KUKA KRL program: RobotSps.src, robotsps.dat

--- RobotSps.src ---
&ACCESS RVE
&REL 156
&COMMENT Ansteuerung Micromaster Frequenzumrichter
&PARAM EDITMASK = *
&PARAM TEMPLATE = C:\KRC\Roboter\Template\ExpertSubmit
DEF RobotSps( )

;************************************************
;              CNC Robotics Ltd
;              www.cncrobotics.co.uk
;************************************************
;     Contact: helpdesk@cncrobotics.co.uk
;     Date: 12/09/23
;     Version: 0.23.48
;************************************************
; Description: sps control specific for the spindle.
;************************************************




IF $T1 THEN
   oMode = 0;
ENDIF
IF $T2 THEN
   oMode = 1;
ENDIF
IF $AUT THEN
   oMode = 2;
ENDIF
IF $EXT THEN
   oMode = 3;
ENDIF

bDoorFault = ($AUT OR $EXT) AND (NOT iDoorSignal)

END

--- robotsps.dat ---
&ACCESS  RV
&COMMENT Ansteuerung Micromaster Frequenzumrichter
&PARAM EDITMASK = *
&PARAM TEMPLATE = C:\KRC\Roboter\Template\ExpertSubmit
&PARAM TEMPLATE = C:\KRC\Roboter\Template\ExpertSubmit
&REL 156
DEFDAT  ROBOTSPS PUBLIC
GLOBAL INT nHeartbeatTime=-1000

;digital inputs

;GLOBAL SIGNAL iDrivesEnabled $IN[] ;drive engage from Pilz mapped directly by Auto External;
;GLOBAL SIGNAL iAcknowledgeMessages $IN[] ;Acknowledge messages from Pilz mapped directly by Auto External
;GLOBAL SIGNAL iStart $IN[] ;operator start button
;GLOBAL SIGNAL iStop $IN[] ;operator stop button
;
;GLOBAL SIGNAL oTeach $OUT[] ;T1 active to Pilz


GLOBAL ENUM SYSTEM_STATE EMERGENCY_STOP,DOOR_OPEN,FAULT,SYSTEM_OK,DRIVES_ON
DECL GLOBAL SYSTEM_STATE systemState=#SYSTEM_OK
DECL GLOBAL STATE_T E_stat
DECL GLOBAL MODUS_T E_mode
GLOBAL BOOL bDoorFault=FALSE
GLOBAL BOOL bRobotHomed=TRUE

ENDDAT
